{attribute 'GeneratedUsingTerminal: KL8610-0003'}
{attribute addProperty BoxType "KL8610-0003"}
{attribute addProperty Description ""}
{attribute addProperty Physics ""}
{attribute addProperty Id "KL8601_1AT %Q*KL_6576A6810KL8601_2AT %Q*KL_6576A6810KL8601_3AT %Q*KL_6576A6810KL8601_4AT %Q*KL_6576A6810"}
{attribute addProperty CRC "1954933029"}
{attribute addProperty Size "0"}
TYPE KL_7485E925 :
STRUCT
	{attribute addProperty Name "KL8601_1"}
	KL8601_1 : KL_6576A681;
	{attribute addProperty Name "KL8601_2"}
	KL8601_2 : KL_6576A681;
	{attribute addProperty Name "KL8601_3"}
	KL8601_3 : KL_6576A681;
	{attribute addProperty Name "KL8601_4"}
	KL8601_4 : KL_6576A681;
END_STRUCT
END_TYPE

(* stored: Version 1.2.0.0, ProductVersion 3.1.4024.9
   DUT KL_7485E925: Id {fbef74c4-59ab-424d-8149-4feb0a65e67c} *)
